TYPE ST_MeasurementVoltageData EXTENDS ST_MeasurementFieldData:
STRUCT
	e_ACrotationStatus		:	eACRotationState;
	ar_PhaseVoltage			: 	ARRAY[0..3] OF REAL;
	ar_LineVoltage			:	ARRAY[0..3] OF REAL;
	li_TimeVoltZeroCrossup 	: 	LINT;
	ar_Frequency			: 	ARRAY[0..3] OF REAL;
	r_VoltageUnbalance		: 	REAL;	
END_STRUCT
END_TYPE

(* stored: Version 1.1.0.1, ProductVersion 3.1.4024.12
   DUT ST_MeasurementVoltageData: Id {ea032aac-7c32-46dd-9283-7e1b9d3b84d4} *)
